Universal Robots PolyScope program: test_gripper.urp

ProgramRoot setBeforeStartSequence=true; setInitialVariableValues=true; directory=/programs/robotiq_2f_gripper_programs; kinematics=(a=[0, -0.425, -0.39225, 0, 0, 0], d=[0.08916, 0, 0, 0.10915, 0.09465, 0.0823], alpha=[1.5708, 0, 0, 1.5708, -1.5708, 0], deltaTheta=[0, 0, 0, 0, 0, 0], status=notInitialized); name=test_gripper; robotEnvironmentFileName=default; serialNumberRobot=2013212154
  InitVariables 
  BeforeStart description=COMMAND_SEQUENCE_BEFORE_PROGRAM_START; name=BeforeStart
    Script type=1; scriptFile=/programs/robotiq_2f_gripper_programs/rq_before_start.script
    Script type=1; scriptFile=/programs/robotiq_2f_gripper_programs/rq_script.script
    Assignment assignmentValueSource=0; expr=0; operatorValueType=INTEGER; valueSource=EXPRESSION; variable=0
    Assignment assignmentValueSource=0; expr=0; operatorValueType=INTEGER; valueSource=EXPRESSION; variable=0
    Assignment assignmentValueSource=0; expr=0; operatorValueType=INTEGER; valueSource=EXPRESSION; variable=0
    Assignment assignmentValueSource=0; expr=0; operatorValueType=INTEGER; valueSource=EXPRESSION; variable=0
  MainProgram cartesianAcceleration=1.2; cartesianSpeed=0.25; jointAcceleration=1.3962634015954636; jointSpeed=1.0471975511965976; moveAsFastAsPossible=true; sharedProcessMoveBlendRadius=0.025; featureReference=(installationNameReference=Base); motionType=JOINT_SPACE; runOnlyOneCycle=true
    Assignment assignmentValueSource=0; expr=255; operatorValueType=INTEGER; valueSource=EXPRESSION; variable=255
    Assignment assignmentValueSource=0; expr=255; operatorValueType=INTEGER; valueSource=EXPRESSION; variable=255
    CallSubProgram subProgramNodeToCall=rq_print_driver_version()
    CallSubProgram subProgramNodeToCall=rq_reset()
    CallSubProgram subProgramNodeToCall=rq_activate_and_wait()
    If expr=ExpressionVariableNode≟1; type=IF_NODE
      Popup message=activation succes; type=MESSAGE
    If type=ELSE_NODE
      Popup message=Error on activation; type=MESSAGE
    Wait analogComparison=0; analogInputRange=0; analogValue=0.0; digitalValue=0; selectedAnalogSensor=-1; selectedDigitalSensor=-1; waitTime=1.0; type=TIMER_WAIT
    CallSubProgram subProgramNodeToCall=rq_reset()
    CallSubProgram subProgramNodeToCall=rq_activate()
    While checkConditionInSeperateThread=true; count=0; expr=ExpressionVariableNode≟0; type=LOOP_EXPR; variable=(name=Loop_1, prefersPersistentValue=false, requestANewUniqueName=false)
      Wait analogComparison=0; analogInputRange=0; analogValue=0.0; digitalValue=0; selectedAnalogSensor=-1; selectedDigitalSensor=-1; waitTime=0.1; type=TIMER_WAIT
      CallSubProgram subProgramNodeToCall=rq_is_gripper_activated()
    Assignment assignmentValueSource=0; expr=0; operatorValueType=INTEGER; valueSource=EXPRESSION; variable=255
    Assignment assignmentValueSource=0; expr=0; operatorValueType=INTEGER; valueSource=EXPRESSION; variable=255
    CallSubProgram subProgramNodeToCall=rq_set_force(rq_force)
    CallSubProgram subProgramNodeToCall=rq_set_speed(rq_speed)
    CallSubProgram subProgramNodeToCall=rq_close_and_wait()
    CallSubProgram subProgramNodeToCall=rq_current_pos()
    Script type=0; expressionBranchNode=popup(rq_pos)
    If expr=ExpressionVariableNode≟1; type=IF_NODE
      CallSubProgram subProgramNodeToCall=rq_open_and_wait()
    If expr=ExpressionVariableNode≟1; type=ELSEIF_NODE
      Wait analogComparison=0; analogInputRange=0; analogValue=0.0; digitalValue=0; selectedAnalogSensor=-1; selectedDigitalSensor=-1; waitTime=2.0; type=TIMER_WAIT
      CallSubProgram subProgramNodeToCall=rq_open_and_wait()
    If type=ELSE_NODE
      Popup message=Got an error on closing gripper; type=MESSAGE
    If expr=ExpressionVariableNode≟1; type=IF_NODE
      CallSubProgram subProgramNodeToCall=rq_close()
    If expr=ExpressionVariableNode≟1; type=ELSEIF_NODE
      Wait analogComparison=0; analogInputRange=0; analogValue=0.0; digitalValue=0; selectedAnalogSensor=-1; selectedDigitalSensor=-1; waitTime=2.0; type=TIMER_WAIT
      CallSubProgram subProgramNodeToCall=rq_close()
    If type=ELSE_NODE
      Popup message=Got an error on opening gripper; type=MESSAGE
    While count=0; expr=ExpressionVariableNode≟0; type=LOOP_EXPR; variable=(name=Loop_2, prefersPersistentValue=false, requestANewUniqueName=false)
      Wait analogComparison=0; analogInputRange=0; analogValue=0.0; digitalValue=0; selectedAnalogSensor=-1; selectedDigitalSensor=-1; waitTime=0.1; type=TIMER_WAIT
      CallSubProgram subProgramNodeToCall=rq_is_motion_complete()
    CallSubProgram subProgramNodeToCall=rq_open()
    While count=0; expr=ExpressionVariableNode≟0; type=LOOP_EXPR; variable=(name=Loop_3, prefersPersistentValue=false, requestANewUniqueName=false)
      Wait analogComparison=0; analogInputRange=0; analogValue=0.0; digitalValue=0; selectedAnalogSensor=-1; selectedDigitalSensor=-1; waitTime=0.1; type=TIMER_WAIT
      CallSubProgram subProgramNodeToCall=rq_is_motion_complete()
    Wait analogComparison=0; analogInputRange=0; analogValue=0.0; digitalValue=0; selectedAnalogSensor=-1; selectedDigitalSensor=-1; waitTime=2.0; type=TIMER_WAIT
    Assignment assignmentValueSource=0; expr=175; operatorValueType=INTEGER; valueSource=EXPRESSION; variable=0
    CallSubProgram subProgramNodeToCall=rq_move(rq_pos)
    Wait analogComparison=0; analogInputRange=0; analogValue=0.0; digitalValue=0; selectedAnalogSensor=-1; selectedDigitalSensor=-1; waitTime=2.0; type=TIMER_WAIT
    CallSubProgram subProgramNodeToCall=rq_stop()
    Assignment assignmentValueSource=0; expr=255; operatorValueType=INTEGER; valueSource=EXPRESSION; variable=255
    Assignment assignmentValueSource=0; expr=255; operatorValueType=INTEGER; valueSource=EXPRESSION; variable=255
    CallSubProgram subProgramNodeToCall=rq_set_force(rq_force)
    CallSubProgram subProgramNodeToCall=rq_set_speed(rq_speed)
    CallSubProgram subProgramNodeToCall=rq_close_and_wait()
    If expr=ExpressionVariableNode≟1; type=IF_NODE
      Popup message=Got object; type=MESSAGE
    If type=ELSE_NODE
      Wait analogComparison=0; analogInputRange=0; analogValue=0.0; digitalValue=0; selectedAnalogSensor=-1; selectedDigitalSensor=-1; waitTime=5.0; type=TIMER_WAIT
    CallSubProgram subProgramNodeToCall=rq_move_and_wait(167)
    CallSubProgram subProgramNodeToCall=rq_move_and_wait(115)
    CallSubProgram subProgramNodeToCall=rq_move_and_wait(65)
    CallSubProgram subProgramNodeToCall=rq_move(167)
    While count=0; expr=ExpressionVariableNode≟0; type=LOOP_EXPR; variable=(name=Loop_4, prefersPersistentValue=false, requestANewUniqueName=false)
      Wait analogComparison=0; analogInputRange=0; analogValue=0.0; digitalValue=0; selectedAnalogSensor=-1; selectedDigitalSensor=-1; waitTime=0.1; type=TIMER_WAIT
      CallSubProgram subProgramNodeToCall=rq_is_motion_complete()
    CallSubProgram subProgramNodeToCall=rq_move(115)
    While count=0; expr=ExpressionVariableNode≟0; type=LOOP_EXPR; variable=(name=Loop_5, prefersPersistentValue=false, requestANewUniqueName=false)
      Wait analogComparison=0; analogInputRange=0; analogValue=0.0; digitalValue=0; selectedAnalogSensor=-1; selectedDigitalSensor=-1; waitTime=0.1; type=TIMER_WAIT
      CallSubProgram subProgramNodeToCall=rq_is_motion_complete()
    CallSubProgram subProgramNodeToCall=rq_move(65)
    While count=0; expr=ExpressionVariableNode≟0; type=LOOP_EXPR; variable=(name=Loop_6, prefersPersistentValue=false, requestANewUniqueName=false)
      Wait analogComparison=0; analogInputRange=0; analogValue=0.0; digitalValue=0; selectedAnalogSensor=-1; selectedDigitalSensor=-1; waitTime=0.1; type=TIMER_WAIT
      CallSubProgram subProgramNodeToCall=rq_is_motion_complete()
    CallSubProgram subProgramNodeToCall=rq_auto_release_open_and_wait()
    CallSubProgram subProgramNodeToCall=rq_print_driver_state()
    CallSubProgram subProgramNodeToCall=rq_print_fault_code()
    CallSubProgram subProgramNodeToCall=rq_print_firmware_version()
    CallSubProgram subProgramNodeToCall=rq_print_num_cycles()
    Wait analogComparison=0; analogInputRange=0; analogValue=0.0; digitalValue=0; selectedAnalogSensor=-1; selectedDigitalSensor=-1; waitTime=5.0; type=TIMER_WAIT
    CallSubProgram subProgramNodeToCall=rq_print_probleme_connection()
  subProgramToCall [hidden by the author, left out]
  subProgramToCall [hidden by the author, left out]
  SubProgram [hidden by the author, left out]
  subProgramToCall [hidden by the author, left out]
  subProgramToCall [hidden by the author, left out]
  subProgramToCall [hidden by the author, left out]
  subProgramToCall [hidden by the author, left out]
  subProgramToCall [hidden by the author, left out]
  subProgramToCall [hidden by the author, left out]
  SubProgram [hidden by the author, left out]
  subProgramToCall [hidden by the author, left out]
  SubProgram [hidden by the author, left out]
  subProgramToCall [hidden by the author, left out]
  subProgramToCall [hidden by the author, left out]
  subProgramToCall [hidden by the author, left out]
  subProgramToCall [hidden by the author, left out]
  subProgramToCall [hidden by the author, left out]
  subProgramToCall [hidden by the author, left out]
  subProgramToCall [hidden by the author, left out]
  subProgramToCall [hidden by the author, left out]
  subProgramToCall [hidden by the author, left out]
  subProgramToCall [hidden by the author, left out]
  subProgramToCall [hidden by the author, left out]
  subProgramToCall [hidden by the author, left out]
  subProgramToCall [hidden by the author, left out]
  subProgramToCall [hidden by the author, left out]
  subProgramToCall [hidden by the author, left out]
  subProgramToCall [hidden by the author, left out]
  subProgramToCall [hidden by the author, left out]
  subProgramToCall [hidden by the author, left out]
